{attribute 'GeneratedUsingTerminal: EP1816-3008-0016'}
{attribute addProperty BoxType "EP1816-3008-0016"}
{attribute addProperty Id "ErrorBOOL1TxPDO_ToggleBOOL1"}
{attribute addProperty CRC "2745852447"}
{attribute addProperty Size "2"}
TYPE Status_A3AA621F :
STRUCT
	{attribute addProperty Name "Error"}
	Error : BOOL;
	{attribute addProperty Name "TxPDO_Toggle"}
	TxPDO_Toggle : BOOL;
END_STRUCT
END_TYPE

(* stored: Version 1.2.0.0, ProductVersion 3.1.4024.9
   DUT Status_A3AA621F: Id {1030ec0b-586e-46c7-8112-87448992e2d4} *)
